{attribute addProperty BoxType "AT2050-0500-0018"}
{attribute addProperty Id "A_0095_AT2021_5250_0019_AT2021_5250AT2021_C5E5984862678.25"}
{attribute addProperty CRC "2778176557"}
{attribute addProperty SizeInBites "626"}
{attribute addProperty SizeInBytes "78.25"}
TYPE A_0049_AT2050_0500_0018_A5979C2D EXTENDS AT2050_BA5A9548 :
STRUCT
	{attribute addProperty Name "A_0095_AT2021_5250_0019_AT2021_5250"}
	A_0095_AT2021_5250_0019_AT2021_5250 : AT2021_C5E59848;
END_STRUCT
END_TYPE

(* stored: Version 1.2.0.0, ProductVersion 3.1.4024.9
   DUT A_0049_AT2050_0500_0018_A5979C2D: Id {3a4f1229-5a08-46a7-8d7d-a5a33b203e1b} *)
